// TwinCAT 3 PLC project PLC_FilterSample
// ProgramVersion: 3.1.4023.0
// libraries:
//   Tc2_Standard, * (Beckhoff Automation GmbH)
//   Tc2_System, * (Beckhoff Automation GmbH)
//   Tc2_Utilities, * (Beckhoff Automation GmbH)
//   Tc3_EventLogger, * (Beckhoff Automation GmbH)
//   Tc3_Module, * (Beckhoff Automation GmbH)
// project tree:
//   / PlcTask.TcTTO
//   POUs/ MAIN.TcPOU, Sample_ClearLoggedEvents.TcPOU, Sample_ExportFilter.TcPOU, Sample_ListenerFilter.TcPOU, FB_SampleListener.TcPOU
// real-time tasks:
//   TASK PlcTask: cycle T#10ms, priority 20, ADS port 350
//   TASK Task 4: cycle T#10ms, priority 1, ADS port 351
//   TASK Task 5: cycle T#10ms, priority 2, ADS port 301

CONFIGURATION PLC_FilterSample
    RESOURCE PLC ON TwinCAT3
        TASK PlcTask(INTERVAL := T#10ms, PRIORITY := 20);
        PROGRAM MAIN WITH PlcTask : MAIN;
    END_RESOURCE
END_CONFIGURATION

// ---- POUs/MAIN.TcPOU
PROGRAM MAIN
VAR
	hr: HRESULT;
	
	bSendEvents: BOOL;
	fbEventLogger : FB_TcEventLogger;
	fbAlarm : FB_TcAlarm; 
	fbSrcInfo : FB_TcSourceInfo; 
END_VAR

Sample_ListenerFilter(); 

//send some events which are used in different filter scenarios 
IF bSendEvents THEN 
	bSendEvents := FALSE; 
	//3 events from one EventClass
	hr := fbEventLogger.SendMessage(TC_EVENTS.TestFilterClass.Event1.uuidEventClass, TC_EVENTS.TestFilterClass.Event1.nEventId, TC_EVENTS.TestFilterClass.Event1.eSeverity, 0,0,0);
	hr := fbEventLogger.SendMessage(TC_EVENTS.TestFilterClass.Event2.uuidEventClass, TC_EVENTS.TestFilterClass.Event2.nEventId, TC_EVENTS.TestFilterClass.Event2.eSeverity, 0,0,0);
	hr := fbEventLogger.SendMessage(TC_EVENTS.TestFilterClass.Event3.uuidEventClass, TC_EVENTS.TestFilterClass.Event3.nEventId, TC_EVENTS.TestFilterClass.Event3.eSeverity, 0,0,0);
	//2 events from another EventClass
	hr := fbEventLogger.SendMessage(TC_EVENTS.TestFilterClass2.EventA.uuidEventClass, TC_EVENTS.TestFilterClass2.EventA.nEventId, TC_EVENTS.TestFilterClass2.EventA.eSeverity, 0,0,0);
	hr := fbEventLogger.SendMessage(TC_EVENTS.TestFilterClass2.EventB.uuidEventClass, TC_EVENTS.TestFilterClass2.EventB.nEventId, TC_EVENTS.TestFilterClass2.EventB.eSeverity, 0,0,0);
	//1 alarm from a 3rd EventClass. Toggle Raise <-> Clear
	fbSrcInfo.sName := 'My Source'; 	
	hr := fbAlarm.Create(TC_EVENTS.MessageTest.Alarm.uuidEventClass, TC_EVENTS.MessageTest.Alarm.nEventId, TC_EVENTS.MessageTest.Alarm.eSeverity, FALSE, fbSrcInfo); 
	hr := fbAlarm.Raise(0);
	//1 message from this EventClass 	
	hr := fbEventLogger.SendMessage(TC_EVENTS.MessageTest.Message.uuidEventClass, TC_EVENTS.MessageTest.Message.nEventId, TC_EVENTS.MessageTest.Message.eSeverity, 0,0,0);
END_IF

Sample_ClearLoggedEvents();

Sample_ExportFilter();

END_PROGRAM

// ---- POUs/Sample_ListenerFilter.TcPOU
// sample about how to set a filter for an event listener
PROGRAM Sample_ListenerFilter
VAR
	hr : HRESULT;
	
	fbMessageListener			: FB_SampleListener;	
	fbListenerFilter			: FB_TcEventFilter; 
	bSubscribeEtherCAT			: BOOL;
	bSubscribeProjectEventClass	: BOOL := TRUE;
	bSubscribed					: BOOL ;
	bUnSubscribe				: BOOL;
END_VAR

fbMessageListener.Execute(); 

//configure the listener to only retrieve 3 events when MAIN.bSendEvents is raised
IF bSubscribeProjectEventClass THEN	
	bSubscribeProjectEventClass := FALSE;  	
	fbListenerFilter.Clear().IsMessage().AND_OP().EventClass.EqualTo(TC_EVENTS.TestFilterClass.Event1.uuidEventClass);  
	hr := fbMessageListener.Subscribe2(fbListenerFilter);
	bSubscribed := TRUE;
END_IF

//configure the listener to only retrieve events (emergency messages) coming in from EtherCAT devices
IF bSubscribeEtherCAT THEN
	bSubscribeEtherCAT := FALSE;  	
	fbListenerFilter.Clear().EtherCATDevice.IsEtherCATDevice(); 
	hr := fbMessageListener.Subscribe2(fbListenerFilter);
	bSubscribed := TRUE;
END_IF

IF bUnSubscribe THEN 
	bUnSubscribe := FALSE; 
	hr := fbMessageListener.Unsubscribe();
	bSubscribed := FALSE;
END_IF

END_PROGRAM

// ---- POUs/FB_SampleListener.TcPOU
FUNCTION_BLOCK FB_SampleListener EXTENDS FB_ListenerBase2

VAR
	nMessages: INT;
END_VAR

METHOD OnMessageSent : HRESULT
VAR_INPUT
	fbEvent : REFERENCE TO FB_TcEvent; 
END_VAR
nMessages := nMessages + 1;
END_METHOD

END_FUNCTION_BLOCK

// ---- POUs/Sample_ClearLoggedEvents.TcPOU
// sample about how to clear filtered logged events
PROGRAM Sample_ClearLoggedEvents
VAR
	hr : HRESULT;
	
	bClear					: BOOL;
	fbClearFilter			: FB_TcEventFilter;
	fbClearLoggedEvents		: FB_TcClearLoggedEventsSettings;
	
	fbEventLogger	: FB_TcEventLogger;
	fbTrig			: R_TRIG;
END_VAR

//this deletes all events with 'TestFilterClass2' eventclass from database (2 per raise on bSendEvents)
fbTrig(CLK:=bClear);
IF bClear THEN
	IF fbTrig.Q THEN
		fbClearFilter.Clear().IsMessage().AND_OP().EventClass.EqualTo(TC_EVENTS.TestFilterClass2.EventA.uuidEventClass); 
		fbClearLoggedEvents.AddFilter(fbClearFilter);
 	END_IF
	IF fbEventLogger.ClearLoggedEvents(fbClearLoggedEvents, hrErrorCode=>hr) THEN // async request returns TRUE if not any more busy
		bClear := FALSE;
	END_IF
END_IF

END_PROGRAM

// ---- POUs/Sample_ExportFilter.TcPOU
// sample about how to export filtered logged events
PROGRAM Sample_ExportFilter
VAR
	hr : HRESULT;
	
	bExport				: BOOL;
	fbCsvExportSetting	: FB_TcEventCsvExportSettings; 
	fbExportFilter		: FB_TcEventFilter; 
	sExportFileName		: STRING := 'c:\temp\Eventlogger-export.csv';
	
	fbEventLogger	: FB_TcEventLogger;
	fbTrig			: R_TRIG;
END_VAR

//this exports the messages with 'MessageTest' eventclass but not the alarms
fbTrig(CLK:=bExport);
IF bExport THEN
	IF fbTrig.Q THEN 
		fbCsvExportSetting.Clear();
		fbCsvExportSetting.AddLanguage(TcLcid.de_DE, 'German');
		fbCsvExportSetting.AddFilter(fbExportFilter); 
		fbExportFilter.Clear().IsMessage().AND_OP().EventClass.EqualTo(TC_EVENTS.MessageTest.Message.uuidEventClass);
	END_IF
	IF fbEventLogger.ExportLoggedEvents(sExportFileName, fbCsvExportSetting, hrErrorCode=>hr) THEN // async request returns TRUE if not any more busy 
		bExport := FALSE;
	END_IF
END_IF

END_PROGRAM
